INTERFACE I_HE_SolidAttenuatorSlot EXTENDS I_Fallible


METHOD GetCenterPosition
VAR_INPUT
    CenterPosition : I_QuantityLREALPublic;
END_VAR
END_METHOD


METHOD GetLength
VAR_INPUT
    Length : I_QuantityLREALPublic;
END_VAR
END_METHOD


METHOD GetMaterial
VAR_IN_OUT
    Material : T_MaxString;
END_VAR
END_METHOD


METHOD GetState : E_HE_SolidAttenuatorSlotState
END_METHOD


METHOD GetThicknessAt
VAR_INPUT
    QueryPointInAxisCoordinates : I_QuantityLREAL;
    Thickness : I_QuantityLREALPublic;
END_VAR
END_METHOD


METHOD HasSpecifiedFilter : BOOL
VAR_INPUT
    Filter : I_HE_SolidAttenuatorFilter;
END_VAR
END_METHOD


METHOD IsEnabled : BOOL
END_METHOD

END_INTERFACE

(* stored: Version 1.1.0.1
   Itf I_HE_SolidAttenuatorSlot: Id {3e8eeb75-9916-40f0-88b6-19addd7d485a}
   Method GetCenterPosition: Id {78205785-44e1-4ed3-afae-b705d8b77b5d}
   Method GetLength: Id {fb86d9c1-a43b-47b3-a6d9-79c92ba8b474}
   Method GetMaterial: Id {24854c65-cec0-4921-a4c5-3586e6d76869}
   Method GetState: Id {140499a8-d9f5-418c-ac5f-ee50adf2d1f8}
   Method GetThicknessAt: Id {9ecc5f3d-b8f9-40d0-a6b0-269c8fded543}
   Method HasSpecifiedFilter: Id {d1bf7eb8-81af-44da-a73f-22357072aa32}
   Method IsEnabled: Id {4e1f759c-f599-4a61-9148-d1e107784260} *)
